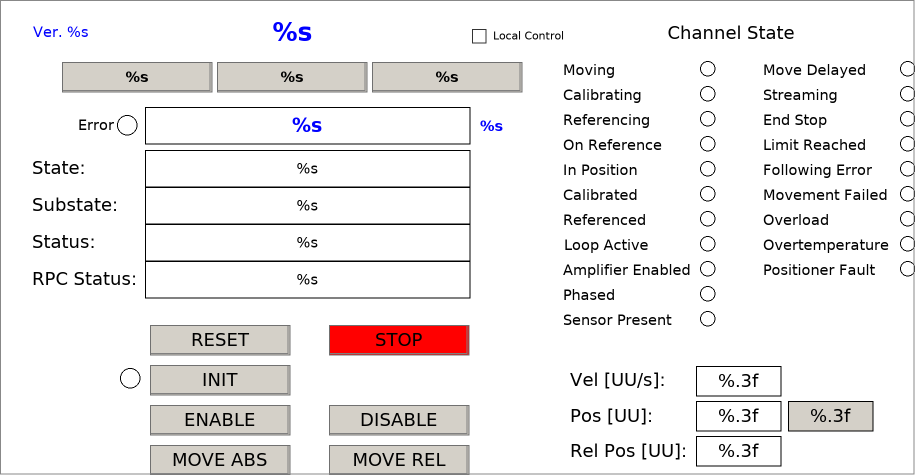
VISUALIZATION GUI_TEMPLATE_SMAR_ACT  // 915x475
VAR_IN_OUT
	m_Instance:	FB_SMAR_ACT_BASE;
END_VAR
    Rectangle (145,107 325x37), "%s", tooltip "Selected Positioner", text variable: m_Instance.ptrGuiCH^.cfg.sName
    Button (62,62 150x30), "%s", tooltip "CH0 Positioner", text variable: m_Instance.arrChName[0]
        OnMouseClick: execute { m_Instance.nGuiIndex := 0; }
    Button (217,62 150x30), "%s", tooltip "CH1 Positioner", text variable: m_Instance.arrChName[1], input disabled if: m_Instance.ptrCH[1] = 0
        OnMouseClick: execute { m_Instance.nGuiIndex := 1; }
    Button (372,62 150x30), "%s", tooltip "CH2 Positioner", text variable: m_Instance.arrChName[2], input disabled if: m_Instance.ptrCH[2] = 0
        OnMouseClick: execute { m_Instance.nGuiIndex := 2; }
    Button (150,365 140x30), "INIT", input disabled if: NOT m_Instance.ptrGuiCH^.stat.bLocal OR m_Instance.ptrGuiCH^.stat.bInitialised
        OnMouseClick: execute { m_Instance.ptrGuiCH^.ctrl.nCmd:=E_SA_CH_CMD.REF; }
    Button (150,445 140x30), "MOVE ABS", input disabled if: NOT m_Instance.ptrGuiCH^.stat.bLocal OR m_Instance.ptrGuiCH^.stat.nState <> E_SA_POS_ELT_STATE.OP
        OnMouseClick: execute { m_Instance.ptrGuiCH^.ctrl.nCmd:=E_SA_CH_CMD.MOV; }
    Rectangle (696,366 85x30), "%.3f", tooltip "Set Velocity [UU/s]", text variable: m_Instance.ptrGuiCH^.ctrl.lrVel
        OnMouseClick: write the text variable via Default
    Label (567,365 100x30), "Vel [UU/s]:"
    Label (567,401 100x30), "Pos [UU]:"
    Rectangle (696,401 85x30), "%.3f", tooltip "Set Position [UU]", text variable: m_Instance.ptrGuiCH^.ctrl.lrPos
        OnMouseClick: write the text variable via Default
    Rectangle (788,401 85x30), "%.3f", tooltip "Actual Position [UU]", text variable: m_Instance.ptrGuiCH^.stat.lrPosActual
    Button (329,325 140x30), "STOP"
        OnMouseClick: execute { m_Instance.ptrGuiCH^.ctrl.nCmd:=E_SA_CH_CMD.STOP; }
    Rectangle (120,12 345x39), "%s", text variable: m_Instance.in_sName
    Label (560,55 140x30), "Moving"
    Label (561,230 140x30), "Loop Active"
    Label (560,80 140x30), "Calibrating"
    Label (560,105 140x30), "Referencing"
    Label (560,305 140x30), "Sensor Present"
    Label (560,180 140x30), "Calibrated"
    Label (560,205 140x30), "Referenced"
    Label (760,105 140x30), "End Stop"
    Label (760,130 140x30), "Limit Reached"
    Label (560,130 140x30), "On Reference"
    Label (560,255 140x30), "Amplifier Enabled"
    Label (560,155 140x30), "In Position"
    Label (75,110 43x30), "Error"
    Ellipse (700,61 15x15), colour toggle: m_Instance.ptrGuiCH^.stat.stState.bACTIVELY_MOVING
    Ellipse (700,236 15x15), colour toggle: m_Instance.ptrGuiCH^.stat.stState.bCLOSED_LOOP_ACTIVE
    Ellipse (700,86 15x15), colour toggle: m_Instance.ptrGuiCH^.stat.stState.bCALIBRATING
    Ellipse (700,111 15x15), colour toggle: m_Instance.ptrGuiCH^.stat.stState.bREFERENCING
    Ellipse (700,311 15x15), colour toggle: m_Instance.ptrGuiCH^.stat.stState.bSENSOR_PRESENT
    Ellipse (700,186 15x15), colour toggle: m_Instance.ptrGuiCH^.stat.stState.bIS_CALIBRATED
    Ellipse (700,211 15x15), colour toggle: m_Instance.ptrGuiCH^.stat.stState.bIS_REFERENCED
    Ellipse (900,111 15x15), colour toggle: m_Instance.ptrGuiCH^.stat.stState.bEND_STOP_REACHED
    Ellipse (900,136 15x15), colour toggle: m_Instance.ptrGuiCH^.stat.stState.bRANGE_LIMIT_REACHED
    Ellipse (700,136 15x15), colour toggle: m_Instance.ptrGuiCH^.stat.stState.bREFERENCE_MARK
    Ellipse (700,261 15x15), colour toggle: m_Instance.ptrGuiCH^.stat.stState.bAMPLIFIER_ENABLED
    Ellipse (700,161 15x15), colour toggle: m_Instance.ptrGuiCH^.stat.stState.bIN_POSITION
    Ellipse (117,115 20x20), colour toggle: m_Instance.ptrGuiCH^.stat.bError
    Label (760,155 140x30), "Following Error"
    Ellipse (900,161 15x15), colour toggle: m_Instance.ptrGuiCH^.stat.stState.bFOLLOWING_LIMIT_REACHED
    Label (760,180 140x30), "Movement Failed"
    Ellipse (900,186 15x15), colour toggle: m_Instance.ptrGuiCH^.stat.stState.bMOVEMENT_FAILED
    Label (760,80 140x30), "Streaming"
    Ellipse (900,86 15x15), colour toggle: m_Instance.ptrGuiCH^.stat.stState.bIS_STREAMING
    Label (760,205 140x30), "Overload"
    Ellipse (900,211 15x15), colour toggle: m_Instance.ptrGuiCH^.stat.stState.bPOSITIONER_OVERLOAD
    Label (760,230 140x30), "Overtemperature"
    Ellipse (900,236 15x15), colour toggle: m_Instance.ptrGuiCH^.stat.stState.bOVER_TEMPERATURE
    Label (560,280 140x30), "Phased"
    Ellipse (700,286 15x15), colour toggle: m_Instance.ptrGuiCH^.stat.stState.bIS_PHASED
    Label (760,255 140x30), "Positioner Fault"
    Ellipse (900,261 15x15), colour toggle: m_Instance.ptrGuiCH^.stat.stState.bPOSITIONER_FAULT
    Label (760,55 140x30), "Move Delayed"
    Ellipse (900,61 15x15), colour toggle: m_Instance.ptrGuiCH^.stat.stState.bMOVE_DELAYED
    Ellipse (120,368 20x20), tooltip "GREEN if initialised", colour toggle: m_Instance.ptrGuiCH^.stat.bInitialised
    Rectangle (145,224 325x37), "%s", tooltip "Positioner Status", text variable: m_Instance.ptrGuiCH^.stat.sStatus
    Rectangle (145,150 325x37), "%s", tooltip "Positioner Device State", text variable: m_Instance.ptrGuiCH^.stat.sState
    Rectangle (145,187 325x37), "%s", tooltip "Positioner Device Substate", text variable: m_Instance.ptrGuiCH^.stat.sSubstate
    Label (29,153 110x30), "State:"
    Label (29,190 110x30), "Substate:"
    Label (29,227 110x30), "Status:"
    Rectangle (30,17 90x30), "Ver. %s", tooltip "SmarAct Library Version", text variable: m_Instance.stat.sLibVersion
    Label (633,18 196x30), "Channel State"
    Rectangle (477,111 59x30), "%s", tooltip "Positioner User Units", text variable: m_Instance.ptrGuiCH^.cfg.sUnits
    Checkbox (470,21 116x30), "Local Control", variable: m_Instance.ptrGuiCH^.stat.bLocal
    Rectangle (145,261 325x37), "%s", tooltip "Positioner Status", text variable: m_Instance.ptrGuiCH^.stat.sRpcErrorText
    Label (29,264 110x30), "RPC Status:"
    Button (150,325 140x30), "RESET", input disabled if: NOT m_Instance.ptrGuiCH^.stat.bLocal
        OnMouseClick: execute { m_Instance.ptrGuiCH^.ctrl.nCmd:=E_SA_CH_CMD.RESET; }
    Label (567,436 130x30), "Rel Pos [UU]:"
    Rectangle (696,436 85x30), "%.3f", tooltip "Set Position Offset [UU]", text variable: m_Instance.ptrGuiCH^.ctrl.lrOff
        OnMouseClick: write the text variable via Default
    Button (329,445 140x30), "MOVE REL", input disabled if: NOT m_Instance.ptrGuiCH^.stat.bLocal OR m_Instance.ptrGuiCH^.stat.nState <> E_SA_POS_ELT_STATE.OP
        OnMouseClick: execute { m_Instance.ptrGuiCH^.ctrl.lrPos := m_Instance.ptrGuiCH^.stat.lrPosActual + m_Instance.ptrGuiCH^.ctrl.lrOff; m_Instance.ptrGuiCH^.ctrl.nCmd:=E_SA_CH_CMD.MOV; }
    Button (150,405 140x30), "ENABLE", input disabled if: NOT m_Instance.ptrGuiCH^.stat.bLocal or NOT m_Instance.ptrGuiCH^.stat.bInitialised OR m_Instance.ptrGuiCH^.stat.nState = E_SA_POS_ELT_STATE.OP
        OnMouseClick: execute { m_Instance.ptrGuiCH^.ctrl.nCmd:=E_SA_CH_CMD.ENABLE; }
    Button (329,405 140x30), "DISABLE", input disabled if: NOT m_Instance.ptrGuiCH^.stat.bLocal OR m_Instance.ptrGuiCH^.stat.nState <> E_SA_POS_ELT_STATE.OP
        OnMouseClick: execute { m_Instance.ptrGuiCH^.ctrl.nCmd:=E_SA_CH_CMD.DISABLE; }
END_VISUALIZATION

(* stored: Version 1.1.0.1, ProductVersion 3.1.4024.10
   Visu GUI_TEMPLATE_SMAR_ACT: Id {8cdc2e82-6967-4e76-9c93-ee4ded37f8d1} *)
